// TIA Portal V19 export
DATA_BLOCK "DB_Zaehler"   // DB80
{ S7_Optimized_Access := 'FALSE' }
AUTHOR : KHE_RE
NAME : DB_LADUN
VERSION : 2.0
// stored: AutoNumber false
   VAR RETAIN
      Anz_Beck : Int := 2;   // wird aus DB1 übernommen
      Offset : Int := 40;   // * Beginn Daten
      leng_Pos : Int := 40;   // * Länge Daten
      Tag_neu : Bool := FALSE;
      Wo_neu : Bool := FALSE;
      Mo_neu : Bool := FALSE;
      res3 : Bool := FALSE;
      res4 : Bool := FALSE;
      res5 : Bool := FALSE;
      res6 : Bool := FALSE;
      AM_Takt : Bool := FALSE;
      I_Time : Byte := 16#01;
      Beck_Nr : Byte := 16#02;
      resb0 : Byte := 16#00;
      MZ_T : Byte := 16#10;   // Merkzelle akt.Tag
      MZ_W : Byte := 16#00;   // Merkzelle akt.Woche
      MZ_M : Byte := 16#06;   // Merkzelle akt.Monat
      Beck_ext : Byte := 16#00;   // Becken-Nr. für externe Dosierzähler
      Wert_Ext : Real := 0.0;   // ext. Zählwert (siehe FC6)
      resDW2 : DWord := 16#0000_0000;
      resDW3 : DWord := 16#0000_0000;
      resDW4 : DWord := 16#0000_0000;
      DosMenge_Typ7 : DWord := 16#0000_0000;
      resDW5 : DWord := 16#0000_0000;
      resW : Word := 16#0000;
      Becken : Array[1..20] of Struct   // * Feldlänge anpassen
         Typ : Byte;   // Typ 0=Ah, 1=Amin, 4=dm2, 6=ext.Zähler(FC6) 8=ext.Ah-Zähler
         Anz_Bad : Byte;   // Anz. des Bäder im Becken
         Input : Array[1..10] of Struct   // Liste der Bäder
            Pos : Int;
         END_STRUCT;
         Zaehl_int : Real;   // interner Restzähler
         Dig_Inp : Byte;   // Dig. Eing. (res.)
         Event : Bool;   // Event Mengenlimit erreicht
         Stop : Bool;   // Dosierzähler gestoppt (von DoPu o.ä.)
         res2 : Bool;
         res3 : Bool;
         res4 : Bool;
         res5 : Bool;
         res6 : Bool;
         Anf_Stp : Bool;   // kumulat.Anforderung Stop DoZa
         resW : Word;
         EventCount : Real;   // Zählzelle für Events
         ext_Val : Real;   // externer Zählwert
         AM_belegt : Word;   // Altmerker Pos.belegt
      END_STRUCT;
   END_VAR
BEGIN
   Becken[1..2].Typ := 16#05;
   Becken[3..20].Typ := 16#00;
   Becken[1..2].Anz_Bad := 16#06;
   Becken[3..20].Anz_Bad := 16#00;
   Becken[1].Input[1].Pos := 1;
   Becken[1].Input[2].Pos := 2;
   Becken[1].Input[3].Pos := 3;
   Becken[1].Input[4].Pos := 4;
   Becken[1].Input[5].Pos := 5;
   Becken[1].Input[6].Pos := 6;
   Becken[1].Input[7..10].Pos := 0;
   Becken[2].Input[1].Pos := 13;
   Becken[2].Input[2].Pos := 14;
   Becken[2].Input[3].Pos := 15;
   Becken[2].Input[4].Pos := 16;
   Becken[2].Input[5].Pos := 17;
   Becken[2].Input[6].Pos := 18;
   Becken[2].Input[7..10].Pos := 0;
   Becken[3].Input[1..10].Pos := 0;
   Becken[4].Input[1..10].Pos := 0;
   Becken[5].Input[1..10].Pos := 0;
   Becken[6].Input[1..10].Pos := 0;
   Becken[7].Input[1..10].Pos := 0;
   Becken[8].Input[1..10].Pos := 0;
   Becken[9].Input[1..10].Pos := 0;
   Becken[10].Input[1..10].Pos := 0;
   Becken[11].Input[1..10].Pos := 0;
   Becken[12].Input[1..10].Pos := 0;
   Becken[13].Input[1..10].Pos := 0;
   Becken[14].Input[1..10].Pos := 0;
   Becken[15].Input[1..10].Pos := 0;
   Becken[16].Input[1..10].Pos := 0;
   Becken[17].Input[1..10].Pos := 0;
   Becken[18].Input[1..10].Pos := 0;
   Becken[19].Input[1..10].Pos := 0;
   Becken[20].Input[1..10].Pos := 0;
   Becken[1..20].Zaehl_int := 0.0;
   Becken[1..20].Dig_Inp := 16#00;
   Becken[1..20].Event := FALSE;
   Becken[1..20].Stop := FALSE;
   Becken[1..20].res2 := FALSE;
   Becken[1..20].res3 := FALSE;
   Becken[1..20].res4 := FALSE;
   Becken[1..20].res5 := FALSE;
   Becken[1..20].res6 := FALSE;
   Becken[1..20].Anf_Stp := FALSE;
   Becken[1..20].resW := 16#0000;
   Becken[1..20].EventCount := 0.0;
   Becken[1..20].ext_Val := 0.0;
   Becken[1..20].AM_belegt := 16#0000;
END_DATA_BLOCK
